KUKA KRL program: wartung.src, wartung.dat

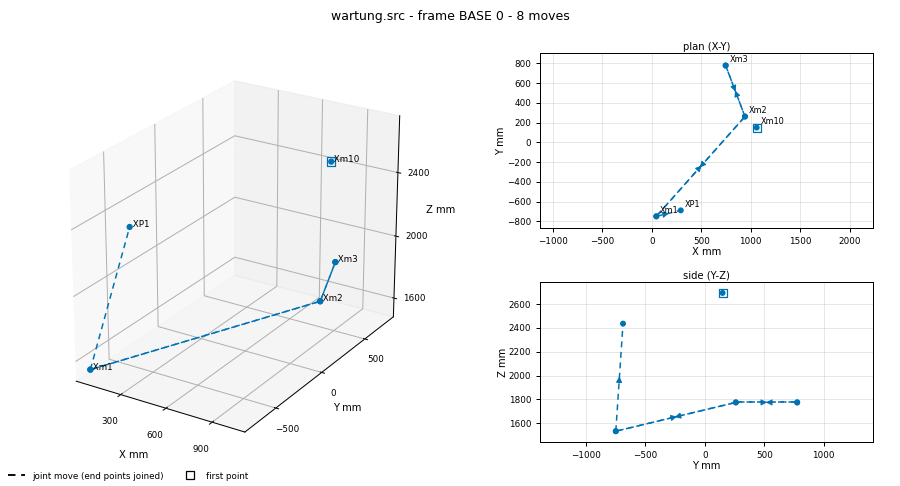
[picture p0: tool path of wartung.src in frame BASE 0, 8 of 11 moves have a stored position in this frame; points joined in program order, loops and branches not executed]
--- wartung.src ---
&ACCESS RVO1
&REL 75
&COMMENT dai_maintence
&USER thsc160
&PARAM DISKPATH = KRC:\R1\Program
&PARAM version = 0.1
DEF wartung( )
;FOLD INI
  ;FOLD BASISTECH INI
    GLOBAL INTERRUPT DECL 3 WHEN $STOPMESS==TRUE DO IR_STOPM ( )
    BAS (#INITMOV,0 )
  ;ENDFOLD (BASISTECH INI)
;FOLD SPOTTECH INI
USERSPOT(#INIT)
;ENDFOLD (SPOTTECH INI)
;FOLD GRIPPERTECH INI
USER_GRP(0,DUMMY,DUMMY,GDEFAULT)
;ENDFOLD (GRIPPERTECH INI)
;FOLD USER INI

;Make your modifications here
;FOLD COLLISION_V_3.01 INI ;%{E}
    IF (COLLISION_DATA[1].I_NR>0) THEN
    GLOBAL INTERRUPT DECL 21 WHEN $IN[COLLISION_DATA[1].I_NR]==FALSE DO COLLSTOP (1,0 )
    ENDIF
    IF (COLLISION_DATA[2].I_NR>0) THEN
    GLOBAL INTERRUPT DECL 22 WHEN $IN[COLLISION_DATA[2].I_NR]==FALSE DO COLLSTOP (2,0 )
    ENDIF
    IF (COLLISION_DATA[3].I_NR>0) THEN
    GLOBAL INTERRUPT DECL 23 WHEN $IN[COLLISION_DATA[3].I_NR]==FALSE DO COLLSTOP (3,0 )
    ENDIF
    IF (COLLISION_DATA[4].I_NR>0) THEN
    GLOBAL INTERRUPT DECL 24 WHEN $IN[COLLISION_DATA[4].I_NR]==FALSE DO COLLSTOP (4,0 )
    ENDIF
;ENDFOLD (Collision)

;ENDFOLD (USER INI)

;ENDFOLD (INI)

; Caracterização dos meios de produção:
; Versão Atual:
; 08/06/2013 12:00 Name: P13.050-R1 CHANGES: Manutenção
; Pinça C2

;FOLD PTP HOME Vel=100 % DEFAULT;%{PE}%R 8.2.20,%MKUKATPBASIS,%CMOVE,%VPTP,%P 1:PTP, 2:HOME, 3:, 5:100, 7:DEFAULT
$BWDSTART=FALSE
PDAT_ACT=PDEFAULT
FDAT_ACT=FHOME
BAS(#PTP_PARAMS,100)
$H_POS=XHOME
PTP XHOME
;ENDFOLD
;FOLD PTP m10 Vel=100 % PDAT19 Tool[8]:TOOL_CHANGER Base[0];%{PE}%R 8.2.20,%MKUKATPBASIS,%CMOVE,%VPTP,%P 1:PTP, 2:m10, 3:, 5:100, 7:PDAT19
$BWDSTART=FALSE
PDAT_ACT=PPDAT19
FDAT_ACT=Fm10
BAS(#PTP_PARAMS,100)
PTP Xm10
;ENDFOLD

chk_w8_wechs_ok ()
wkz1_an ()

;FOLD PTP HOME1 Vel=100 % DEFAULT;%{PE}%R 8.2.20,%MKUKATPBASIS,%CMOVE,%VPTP,%P 1:PTP, 2:HOME1, 3:, 5:100, 7:DEFAULT
$BWDSTART=FALSE
PDAT_ACT=PDEFAULT
FDAT_ACT=FHOME1
BAS(#PTP_PARAMS,100)
PTP XHOME1
;ENDFOLD
;FOLD PTP m1 CONT Vel=100 % PDAT8 Tool[1]:GUN X1 Base[0];%{PE}%R 8.2.20,%MKUKATPBASIS,%CMOVE,%VPTP,%P 1:PTP, 2:m1, 3:C_DIS, 5:100, 7:PDAT8
$BWDSTART=FALSE
PDAT_ACT=PPDAT8
FDAT_ACT=Fm1
BAS(#PTP_PARAMS,100)
PTP Xm1 C_DIS
;ENDFOLD
;FOLD PTP m2 CONT Vel=100 % PDAT11 Tool[1]:GUN X1 Base[0];%{PE}%R 8.2.20,%MKUKATPBASIS,%CMOVE,%VPTP,%P 1:PTP, 2:m2, 3:C_DIS, 5:100, 7:PDAT11
$BWDSTART=FALSE
PDAT_ACT=PPDAT11
FDAT_ACT=Fm2
BAS(#PTP_PARAMS,100)
PTP Xm2 C_DIS
;ENDFOLD
;FOLD PTP m3 CONT Vel=100 % PDAT12 Tool[1]:GUN X1 Base[0];%{PE}%R 8.2.20,%MKUKATPBASIS,%CMOVE,%VPTP,%P 1:PTP, 2:m3, 3:C_DIS, 5:100, 7:PDAT12
$BWDSTART=FALSE
PDAT_ACT=PPDAT12
FDAT_ACT=Fm3
BAS(#PTP_PARAMS,100)
PTP Xm3 C_DIS
;ENDFOLD

;FOLD ; Ponto de Manutencao;%{PE}%R 8.2.20,%MKUKATPBASIS,%CCOMMENT,%VNORMAL,%P 2:Ponto  de  Manutencao
;ENDFOLD
;FOLD PTP Maintenance Vel=100 % PDAT10;%{PE}%R 8.2.20,%MKUKATPBASIS,%CMOVE,%VPTP,%P 1:PTP, 2:Maintenance, 3:, 5:100, 7:PDAT10
$BWDSTART=FALSE
PDAT_ACT=PPDAT10
FDAT_ACT=FMaintenance
BAS(#PTP_PARAMS,100)
PTP XMaintenance
;ENDFOLD

MSG_SHOW("DAI_H_Prog",#notify,999,"dai_maintenance_0")
;FOLD OUT 3218 'WPER:Wartungspos. erreicht'  State= TRUE ;%{PE}%R 5.2.22,%MKUKATPBASIS,%COUT,%VOUTX,%P 2:3218, 3:WPER:Wartungspos. erreicht, 5:TRUE, 6:
    $OUT[3218]=TRUE
;ENDFOLD
Halt
;FOLD WAIT FOR ( NOT IN 3218 'ANFWP:Anforderung Wartungspos.' );%{PE}%R 5.2.22,%MKUKATPBASIS,%CEXT_WAIT_FOR,%VEXT_WAIT_FOR,%P 2:, 4:NOT, 5:$IN, 6:3218, 7:ANFWP:Anforderung Wartungspos., 9:
    WAIT FOR  (  NOT $IN[3218] )
;ENDFOLD
;FOLD OUT 3218 'WPER:Wartungspos. erreicht'  State= FALSE ;%{PE}%R 5.2.22,%MKUKATPBASIS,%COUT,%VOUTX,%P 2:3218, 3:WPER:Wartungspos. erreicht, 5:FALSE, 6:
    $OUT[3218]=FALSE
;ENDFOLD

;FOLD PTP m7 CONT Vel=100 % PDAT16 Tool[1]:GUN X1 Base[0];%{PE}%R 8.2.20,%MKUKATPBASIS,%CMOVE,%VPTP,%P 1:PTP, 2:m7, 3:C_DIS, 5:100, 7:PDAT16
$BWDSTART=FALSE
PDAT_ACT=PPDAT16
FDAT_ACT=Fm7
BAS(#PTP_PARAMS,100)
PTP Xm7 C_DIS
;ENDFOLD
;FOLD PTP m8 CONT Vel=100 % PDAT17 Tool[1]:GUN X1 Base[0];%{PE}%R 8.2.20,%MKUKATPBASIS,%CMOVE,%VPTP,%P 1:PTP, 2:m8, 3:C_DIS, 5:100, 7:PDAT17
$BWDSTART=FALSE
PDAT_ACT=PPDAT17
FDAT_ACT=Fm8
BAS(#PTP_PARAMS,100)
PTP Xm8 C_DIS
;ENDFOLD
;FOLD PTP m9 CONT Vel=100 % PDAT18 Tool[1]:GUN X1 Base[0];%{PE}%R 8.2.20,%MKUKATPBASIS,%CMOVE,%VPTP,%P 1:PTP, 2:m9, 3:C_DIS, 5:100, 7:PDAT18
$BWDSTART=FALSE
PDAT_ACT=PPDAT18
FDAT_ACT=Fm9
BAS(#PTP_PARAMS,100)
PTP Xm9 C_DIS
;ENDFOLD

wkz1_ab ()


;FOLD PTP P1 Vel=100 % PDAT20 Tool[8]:TOOL_CHANGER Base[0];%{PE}%R 8.2.20,%MKUKATPBASIS,%CMOVE,%VPTP,%P 1:PTP, 2:P1, 3:, 5:100, 7:PDAT20
$BWDSTART=FALSE
PDAT_ACT=PPDAT20
FDAT_ACT=FP1
BAS(#PTP_PARAMS,100)
PTP XP1
;ENDFOLD
END

--- wartung.dat ---
&ACCESS RVO1
&REL 75
&COMMENT dai_maintence
&USER thsc160
&PARAM DISKPATH = KRC:\R1\Program
&PARAM version = 0.1
DEFDAT  wartung
;FOLD EXTERNAL DECLARATIONS;%{PE}%MKUKATPBASIS,%CEXT,%VCOMMON,%P
;FOLD GRIPPERTECH EXT
EXT  H50 (INT  :IN,INT  :IN,INT  :IN,GRP_TYP  :IN )
;ENDFOLD (GRIPPERTECH EXT)
;FOLD SPOTTECH EXT
EXT  USERSPOT (S_COMMAND  :IN,SPOT_TYPE  :IN )
;ENDFOLD (SPOTTECH EXT)
;FOLD BASISTECH EXT;%{PE}%MKUKATPBASIS,%CEXT,%VEXT,%P
EXT  BAS (BAS_COMMAND  :IN,REAL  :IN )
DECL INT SUCCESS
;ENDFOLD (BASISTECH EXT)
;FOLD USER EXT;%{E}%MKUKATPUSER,%CEXT,%VEXT,%P
;Make here your modifications
;FOLD COLLISION
EXT  COLLSTOP (INT  :IN,INT  :IN )
;ENDFOLD  (Collision)
;ENDFOLD (USER EXT)
;ENDFOLD (EXTERNAL DECLERATIONS)

DECL BASIS_SUGG_T LAST_BASIS={POINT1[] "P0                      ",POINT2[] "P0                      ",CP_PARAMS[] "CPDAT0                  ",PTP_PARAMS[] "PDAT0                   ",CONT[] "                        ",CP_VEL[] "2.0                     ",PTP_VEL[] "100                     ",SYNC_PARAMS[] "SYNCDAT                 ",SPL_NAME[] "S0                      "}


DECL FDAT FHOME={TOOL_NO 0,BASE_NO 0,IPO_FRAME #BASE}

DECL E6AXIS XMaintenance={A1 -104.496902,A2 -66.4574966,A3 108.875999,A4 -3.08347511,A5 49.5483589,A6 44.7975807,E1 199.958893,E2 0.0,E3 0.0,E4 0.0,E5 0.0,E6 0.0}
DECL FDAT FMaintenance={TOOL_NO 1,BASE_NO 0,IPO_FRAME #BASE,POINT2[] " ",TQ_STATE FALSE}

DECL PDAT PPDAT10={VEL 100.0,ACC 100.0,APO_DIST 100.0}
DECL FDAT FHOME1={TOOL_NO 0,BASE_NO 0,IPO_FRAME #BASE,POINT2[] " ",TQ_STATE FALSE}
DECL PDAT PPDAT8={VEL 100.0,ACC 100.0,APO_DIST 100.0,APO_MODE #CDIS}
DECL E6POS Xm1={X 45.0234604,Y -748.435913,Z 1531.74194,A -86.3570633,B 78.263298,C 69.7170334,S 2,T 2,E1 199.996994,E2 0.0,E3 0.0,E4 0.0,E5 0.0,E6 0.0}
DECL FDAT Fm1={TOOL_NO 1,BASE_NO 0,IPO_FRAME #BASE,POINT2[] " ",TQ_STATE FALSE}
DECL E6POS XM2={X 941.692627,Y 261.335114,Z 1773.974,A 4.78774118,B 68.8631668,C 59.0257988,S 2,T 3,E1 199.995895,E2 0.0,E3 0.0,E4 0.0,E5 0.0,E6 0.0}
DECL FDAT Fm2={TOOL_NO 1,BASE_NO 0,IPO_FRAME #BASE,POINT2[] " ",TQ_STATE FALSE}
DECL PDAT PPDAT11={VEL 100.0,ACC 100.0,APO_DIST 100.0,APO_MODE #CDIS}
DECL E6POS XM3={X 746.397217,Y 777.43573,Z 1773.974,A 38.7877998,B 68.8632507,C 59.0258904,S 2,T 3,E1 199.9953,E2 0.0,E3 0.0,E4 0.0,E5 0.0,E6 0.0}
DECL FDAT Fm3={TOOL_NO 1,BASE_NO 0,IPO_FRAME #BASE,POINT2[] " ",TQ_STATE FALSE}
DECL PDAT PPDAT12={VEL 100.0,ACC 100.0,APO_DIST 100.0,APO_MODE #CDIS}
DECL PDAT PPDAT16={VEL 100.0,ACC 100.0,APO_DIST 100.0,APO_MODE #CDIS}
DECL E6POS Xm7={X 746.396606,Y 777.434998,Z 1773.97302,A 38.7878189,B 68.863327,C 59.0259285,S 2,T 3,E1 199.994705,E2 0.0,E3 0.0,E4 0.0,E5 0.0,E6 0.0}
DECL FDAT Fm7={TOOL_NO 1,BASE_NO 0,IPO_FRAME #BASE,POINT2[] " ",TQ_STATE FALSE}
DECL PDAT PPDAT17={VEL 100.0,ACC 100.0,APO_DIST 100.0,APO_MODE #CDIS}
DECL E6POS Xm8={X 941.692078,Y 261.335205,Z 1773.97302,A 4.78778601,B 68.8632278,C 59.0258484,S 2,T 3,E1 199.995407,E2 0.0,E3 0.0,E4 0.0,E5 0.0,E6 0.0}
DECL FDAT Fm8={TOOL_NO 1,BASE_NO 0,IPO_FRAME #BASE,POINT2[] " ",TQ_STATE FALSE}
DECL PDAT PPDAT18={VEL 100.0,ACC 100.0,APO_DIST 100.0,APO_MODE #CDIS}
DECL E6POS Xm9={X 45.0241814,Y -748.435425,Z 1531.74097,A -86.3570099,B 78.2633591,C 69.7170715,S 2,T 2,E1 199.996597,E2 0.0,E3 0.0,E4 0.0,E5 0.0,E6 0.0}
DECL FDAT Fm9={TOOL_NO 1,BASE_NO 0,IPO_FRAME #BASE,POINT2[] " ",TQ_STATE FALSE}
DECL E6POS XM10={X 1060.198,Y 149.669205,Z 2694.80103,A 40.7707291,B -55.3351593,C 131.170303,S 2,T 11,E1 407.454102,E2 0.0,E3 0.0,E4 0.0,E5 0.0,E6 0.0}
DECL FDAT Fm10={TOOL_NO 8,BASE_NO 0,IPO_FRAME #BASE,POINT2[] " ",TQ_STATE FALSE}
DECL PDAT PPDAT19={VEL 100.0,ACC 100.0,APO_DIST 100.0,APO_MODE #CDIS}
DECL E6POS XP1={X 292.377899,Y -687.815918,Z 2436.698,A -37.667469,B -40.7472115,C 153.499893,S 2,T 10,E1 428.214111,E2 0.0,E3 0.0,E4 0.0,E5 0.0,E6 0.0}
DECL FDAT FP1={TOOL_NO 8,BASE_NO 0,IPO_FRAME #BASE,POINT2[] " ",TQ_STATE FALSE}
DECL PDAT PPDAT20={VEL 100.0,ACC 100.0,APO_DIST 100.0,APO_MODE #CDIS}
ENDDAT
